FUNCTION_BLOCK StructProducer
  (* Standard: 61499-2 *)
  (* Version 1.0, 2026-05-31, Dimitrios Kalligaridis *)
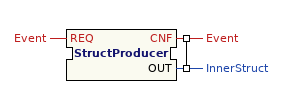
  EVENT_INPUT
    REQ;
  END_EVENT
  EVENT_OUTPUT
    CNF WITH OUT;
  END_EVENT
  VAR_OUTPUT
    OUT : mypackage::InnerStruct;
  END_VAR
END_FUNCTION_BLOCK
